// TIA Portal V20 export
DATA_BLOCK "SP205"   // DB343
// stored: MemoryReserve 100
   VAR
      "PENDANT REQUIRED PL (YELLOW)" : Bool := TRUE;
      SPARE : Bool := FALSE;
      "HOME PBL LAMP ON (GREEN)" : Bool := FALSE;
      SPARE_1 : Bool := FALSE;
      SPARE_2 : Bool := FALSE;
      SPARE_3 : Bool := FALSE;
      SPARE_4 : Bool := FALSE;
      "SCS SELECT DISABLE PL (GREEN)" : Bool := TRUE;
   END_VAR
BEGIN
END_DATA_BLOCK
